FUNCTION_BLOCK "EM_TransferFeed"
{ S7_Optimized_Access := 'TRUE' }
   VAR
      Static : Bool;
   END_VAR

BEGIN

END_FUNCTION_BLOCK
